{attribute 'GeneratedUsingTerminal: KL1501'}
{attribute addProperty BoxType "KL1501"}
{attribute addProperty Id "Channel_1AT %Q*Channel_3C1A65000"}
{attribute addProperty CRC "3994895622"}
{attribute addProperty Size "0"}
TYPE KL1501_EE1D4506 :
STRUCT
	{attribute addProperty Name "Channel_1"}
	Channel_1 : Channel_3C1A6500;
END_STRUCT
END_TYPE

(* stored: Version 1.2.0.0, ProductVersion 3.1.4024.9
   DUT KL1501_EE1D4506: Id {15758f5a-b6b7-4e7f-8eae-fa04fd901881} *)
